PROGRAM MAIN
VAR
END_VAR

END_PROGRAM

(* stored: Version 1.1.0.1
   POU MAIN: Id {1e648042-dba3-4275-8844-6a8a163a0ce7} *)
